{attribute addProperty BoxType "KL9900-0056"}
{attribute addProperty Id "Channel_1Channel_129BF9DC00"}
{attribute addProperty CRC "614033824"}
{attribute addProperty SizeInBites "0"}
{attribute addProperty SizeInBytes "0"}
TYPE KL_249969A0 :
STRUCT
	{attribute addProperty Name "Channel_1"}
	Channel_1 : Channel_129BF9DC;
END_STRUCT
END_TYPE

(* stored: Version 1.2.0.0, ProductVersion 3.1.4024.9
   DUT KL_249969A0: Id {de2ec46e-57cf-4592-a2b3-f211d8fffc02} *)
